FUNCTION_BLOCK Recipe_10054_FreePassion_special
VAR_INPUT
	execute: BOOL;
	Order: DUT_RECIPEORDER;
END_VAR
VAR_OUTPUT
	RecipeInfo: DUT_RECIPEOFFER;
	RecipeDone: BOOL;
	InitDone: BOOL;
END_VAR
VAR
	userparametersum: LREAL;
	StepDone: BOOL;
	i: INT;
END_VAR

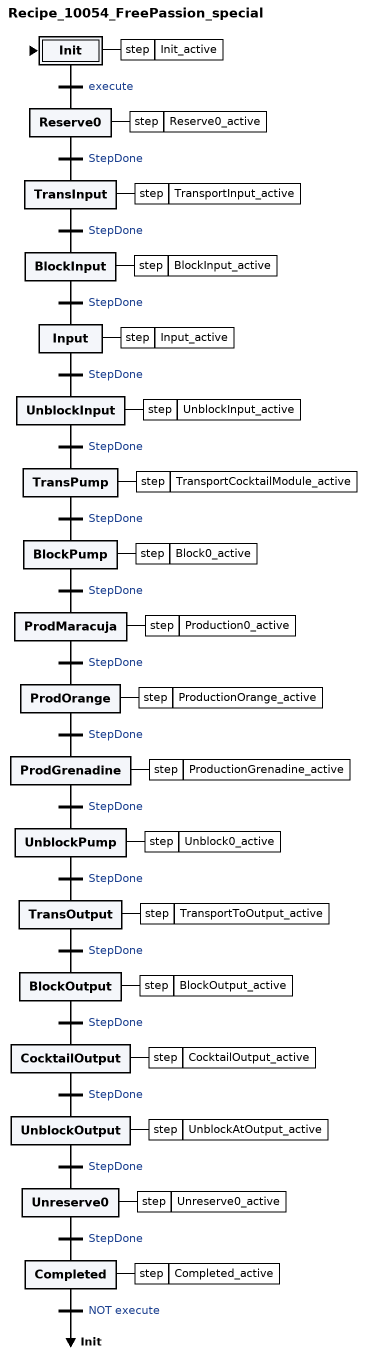
INITIAL_STEP Init:
    Init_active(N);  // step action
END_STEP
TRANSITION FROM Init TO Reserve0
    := execute;
END_TRANSITION
STEP Reserve0:
    Reserve0_active(N);  // step action
END_STEP
TRANSITION FROM Reserve0 TO TransInput
    := StepDone;
END_TRANSITION
STEP TransInput:
    TransportInput_active(N);  // step action
END_STEP
TRANSITION FROM TransInput TO BlockInput
    := StepDone;
END_TRANSITION
STEP BlockInput:
    BlockInput_active(N);  // step action
END_STEP
TRANSITION FROM BlockInput TO Input
    := StepDone;
END_TRANSITION
STEP Input:
    Input_active(N);  // step action
END_STEP
TRANSITION FROM Input TO UnblockInput
    := StepDone;
END_TRANSITION
STEP UnblockInput:
    UnblockInput_active(N);  // step action
END_STEP
TRANSITION FROM UnblockInput TO TransPump
    := StepDone;
END_TRANSITION
STEP TransPump:
    TransportCocktailModule_active(N);  // step action
END_STEP
TRANSITION FROM TransPump TO BlockPump
    := StepDone;
END_TRANSITION
STEP BlockPump:
    Block0_active(N);  // step action
END_STEP
TRANSITION FROM BlockPump TO ProdMaracuja
    := StepDone;
END_TRANSITION
STEP ProdMaracuja:
    Production0_active(N);  // step action
END_STEP
TRANSITION FROM ProdMaracuja TO ProdOrange
    := StepDone;
END_TRANSITION
STEP ProdOrange:
    ProductionOrange_active(N);  // step action
END_STEP
TRANSITION FROM ProdOrange TO ProdGrenadine
    := StepDone;
END_TRANSITION
STEP ProdGrenadine:
    ProductionGrenadine_active(N);  // step action
END_STEP
TRANSITION FROM ProdGrenadine TO UnblockPump
    := StepDone;
END_TRANSITION
STEP UnblockPump:
    Unblock0_active(N);  // step action
END_STEP
TRANSITION FROM UnblockPump TO TransOutput
    := StepDone;
END_TRANSITION
STEP TransOutput:
    TransportToOutput_active(N);  // step action
END_STEP
TRANSITION FROM TransOutput TO BlockOutput
    := StepDone;
END_TRANSITION
STEP BlockOutput:
    BlockOutput_active(N);  // step action
END_STEP
TRANSITION FROM BlockOutput TO CocktailOutput
    := StepDone;
END_TRANSITION
STEP CocktailOutput:
    CocktailOutput_active(N);  // step action
END_STEP
TRANSITION FROM CocktailOutput TO UnblockOutput
    := StepDone;
END_TRANSITION
STEP UnblockOutput:
    UnblockAtOutput_active(N);  // step action
END_STEP
TRANSITION FROM UnblockOutput TO Unreserve0
    := StepDone;
END_TRANSITION
STEP Unreserve0:
    Unreserve0_active(N);  // step action
END_STEP
TRANSITION FROM Unreserve0 TO Completed
    := StepDone;
END_TRANSITION
STEP Completed:
    Completed_active(N);  // step action
END_STEP
TRANSITION FROM Completed TO Init
    := NOT execute;
END_TRANSITION

ACTION Production0_active:
StepDone := FALSE;

userparametersum := 0;
FOR i := 1 TO UserParameterCnt DO
	IF NOT (order.UserParameter[i].Value = 0) THEN
		userparametersum := userparametersum + order.UserParameter[i].Value;
	
	END_IF
END_FOR
IF userparametersum = 0 THEN
userparametersum := -1;
END_IF
//Skill auswählen
ExecuteSkill.SkillID 		:= 1113;
ExecuteSkill.SkillName	 	:= 'Marajuca Juice';

//Parameter setzen

ExecuteSkill.Parameter[0].ID := 1;
ExecuteSkill.Parameter[0].Name := 'Quantity';
//order.userParameter[0] = amount
ExecuteSkill.Parameter[0].Value := order.UserParameter[0].Value * order.UserParameter[1].Value / userparametersum;//Summe aller Zutatenmengen;


(*
ExecuteSkill.Parameter[2].ID := ;
ExecuteSkill.Parameter[2].Name := '';
ExecuteSkill.Parameter[2].Value := ;
*)

(*
ExecuteSkill.Parameter[3].ID := ;
ExecuteSkill.Parameter[3].Name := '';
ExecuteSkill.Parameter[3].Value := ;
*)

(*
ExecuteSkill.Parameter[4].ID := ;
ExecuteSkill.Parameter[4].Name := '';
ExecuteSkill.Parameter[4].Value := ;
*)

(*
ExecuteSkill.Parameter[5].ID := ;
ExecuteSkill.Parameter[5].Name := '';
ExecuteSkill.Parameter[5].Value := ;
*)



ExecuteSkill();

StepDone := ExecuteSkill.Done;
END_ACTION

ACTION TransportInput_active:
StepDone := FALSE;

//Skill auswählen
ExecuteSkill.SkillID 		:= 1320;
ExecuteSkill.SkillName	 	:= 'Transport';

//Parameter setzen

ExecuteSkill.Parameter[3].ID := 3;
ExecuteSkill.Parameter[3].Name := 'Velocity';
ExecuteSkill.Parameter[3].Value := 1500;



ExecuteSkill.Parameter[1].ID :=  1;
ExecuteSkill.Parameter[1].Name := 'TargetPosition X';
ExecuteSkill.Parameter[1].Value := 30 ;
ExecuteSkill.Parameter[1].StringValue := '#DP#2#XPosition';



ExecuteSkill.Parameter[2].ID := 2;
ExecuteSkill.Parameter[2].Name := 'TargetPosition Z';
ExecuteSkill.Parameter[2].Value := 100;// ZCookieModule - ZCookieModuleCalibration - 2* Cookiethickness + toppingthickness+ Preasureheight  ;



(*
ExecuteSkill.Parameter[4].ID := 4;
ExecuteSkill.Parameter[4].Name := 'Acceleration';
ExecuteSkill.Parameter[4].Value := 0 ;
*)

(*
ExecuteSkill.Parameter[5].ID := ;
ExecuteSkill.Parameter[5].Name := '';
ExecuteSkill.Parameter[5].Value := ;
*)



ExecuteSkill();

StepDone := ExecuteSkill.Done;
END_ACTION

ACTION BlockOutput_active:
StepDone := FALSE;

//Skill auswählen
ExecuteSkill.SkillID 		:= 1315;
ExecuteSkill.SkillName	 	:= 'Block';

//Parameter setzen

ExecuteSkill.Parameter[1].ID := 1;
ExecuteSkill.Parameter[1].Name := 'TaskID';
ExecuteSkill.Parameter[1].Value := Order.TaskID;


(*
ExecuteSkill.Parameter[2].ID := ;
ExecuteSkill.Parameter[2].Name := '';
ExecuteSkill.Parameter[2].Value := ;
*)

(*
ExecuteSkill.Parameter[3].ID := ;
ExecuteSkill.Parameter[3].Name := '';
ExecuteSkill.Parameter[3].Value := ;
*)

(*
ExecuteSkill.Parameter[4].ID := ;
ExecuteSkill.Parameter[4].Name := '';
ExecuteSkill.Parameter[4].Value := ;
*)

(*
ExecuteSkill.Parameter[5].ID := ;
ExecuteSkill.Parameter[5].Name := '';
ExecuteSkill.Parameter[5].Value := ;
*)



ExecuteSkill();

StepDone := ExecuteSkill.Done;
END_ACTION

ACTION ProductionGrenadine_active:
StepDone := FALSE;

//Skill auswählen
ExecuteSkill.SkillID 		:= 1121;
ExecuteSkill.SkillName	 	:= 'Batida de Coco';

//Parameter setzen

ExecuteSkill.Parameter[0].ID := 1;
ExecuteSkill.Parameter[0].Name := 'Quantity';
//order.userParameter[0] = amount
ExecuteSkill.Parameter[0].Value := order.UserParameter[0].Value * order.UserParameter[3].Value / userparametersum; //Summe aller Zutatenmengen;



(*
ExecuteSkill.Parameter[2].ID := ;
ExecuteSkill.Parameter[2].Name := '';
ExecuteSkill.Parameter[2].Value := ;
*)

(*
ExecuteSkill.Parameter[3].ID := ;
ExecuteSkill.Parameter[3].Name := '';
ExecuteSkill.Parameter[3].Value := ;
*)

(*
ExecuteSkill.Parameter[4].ID := ;
ExecuteSkill.Parameter[4].Name := '';
ExecuteSkill.Parameter[4].Value := ;
*)

(*
ExecuteSkill.Parameter[5].ID := ;
ExecuteSkill.Parameter[5].Name := '';
ExecuteSkill.Parameter[5].Value := ;
*)



ExecuteSkill();

StepDone := ExecuteSkill.Done;
END_ACTION

ACTION Unreserve0_active:
StepDone := FALSE;

//Skill auswählen
ExecuteSkill.SkillID 		:= 1311;
ExecuteSkill.SkillName	 	:= 'Unreserve';

//Parameter setzen

ExecuteSkill.Parameter[1].ID := 1;
ExecuteSkill.Parameter[1].Name := 'TaskID';
ExecuteSkill.Parameter[1].Value := Order.TaskID;


(*
ExecuteSkill.Parameter[2].ID := ;
ExecuteSkill.Parameter[2].Name := '';
ExecuteSkill.Parameter[2].Val ue := ;
*)

(*
ExecuteSkill.Parameter[3].ID := ;
ExecuteSkill.Parameter[3].Name := '';
ExecuteSkill.Parameter[3].Value := ;
*)

(*
ExecuteSkill.Parameter[4].ID := ;
ExecuteSkill.Parameter[4].Name := '';
ExecuteSkill.Parameter[4].Value := ;
*)

(*
ExecuteSkill.Parameter[5].ID := ;
ExecuteSkill.Parameter[5].Name := '';
ExecuteSkill.Parameter[5].Value := ;
*)



ExecuteSkill();

StepDone := ExecuteSkill.Done;
END_ACTION

ACTION Input_active:
StepDone := FALSE;

//Skill auswählen
ExecuteSkill.SkillID 		:= 1402;
ExecuteSkill.SkillName	 	:= 'Input';

//Parameter setzen

ExecuteSkill.Parameter[1].ID := 1;
ExecuteSkill.Parameter[1].Name := 'TaskID';
ExecuteSkill.Parameter[1].Value := Order.TaskID;


(*
ExecuteSkill.Parameter[2].ID := ;
ExecuteSkill.Parameter[2].Name := '';
ExecuteSkill.Parameter[2].Value := ;
*)

(*
ExecuteSkill.Parameter[3].ID := ;
ExecuteSkill.Parameter[3].Name := '';
ExecuteSkill.Parameter[3].Value := ;
*)

(*
ExecuteSkill.Parameter[4].ID := ;
ExecuteSkill.Parameter[4].Name := '';
ExecuteSkill.Parameter[4].Value := ;
*)

(*
ExecuteSkill.Parameter[5].ID := ;
ExecuteSkill.Parameter[5].Name := '';
ExecuteSkill.Parameter[5].Value := ;
*)



ExecuteSkill();

StepDone := ExecuteSkill.Done;
END_ACTION

ACTION TransportToOutput_active:
StepDone := FALSE;

//Skill auswählen
ExecuteSkill.SkillID 		:= 1320;
ExecuteSkill.SkillName	 	:= 'Transport';

//Parameter setzen

ExecuteSkill.Parameter[3].ID := 3;
ExecuteSkill.Parameter[3].Name := 'Velocity';
ExecuteSkill.Parameter[3].Value := 280;



ExecuteSkill.Parameter[1].ID :=  1;
ExecuteSkill.Parameter[1].Name := 'TargetPosition X';
ExecuteSkill.Parameter[1].Value := 30 ;
ExecuteSkill.Parameter[1].StringValue := '#DP#2#XPosition';



ExecuteSkill.Parameter[2].ID := 2;
ExecuteSkill.Parameter[2].Name := 'TargetPosition Z';
ExecuteSkill.Parameter[2].Value := ZInputOutput;// ZCookieModule - ZCookieModuleCalibration - 2* Cookiethickness + toppingthickness+ Preasureheight  ;



(* ExecuteSkill.Parameter[4].ID := 4;
ExecuteSkill.Parameter[4].Name := 'Acceleration';
ExecuteSkill.Parameter[4].Value :=0 ;

*)
(*
ExecuteSkill.Parameter[5].ID := ;
ExecuteSkill.Parameter[5].Name := '';
ExecuteSkill.Parameter[5].Value := ;
*)



ExecuteSkill();

StepDone := ExecuteSkill.Done;
END_ACTION

ACTION ProductionOrange_active:
StepDone := FALSE;

//Skill auswählen
ExecuteSkill.SkillID 		:= 1117;
ExecuteSkill.SkillName	 	:= 'Orange';

//Parameter setzen

ExecuteSkill.Parameter[0].ID := 1;
ExecuteSkill.Parameter[0].Name := 'Quantity';
//order.userParameter[0] = amount
ExecuteSkill.Parameter[0].Value := order.UserParameter[0].Value * order.UserParameter[2].Value / userparametersum;//Summe aller Zutatenmengen;



(*
ExecuteSkill.Parameter[2].ID := ;
ExecuteSkill.Parameter[2].Name := '';
ExecuteSkill.Parameter[2].Value := ;
*)

(*
ExecuteSkill.Parameter[3].ID := ;
ExecuteSkill.Parameter[3].Name := '';
ExecuteSkill.Parameter[3].Value := ;
*)

(*
ExecuteSkill.Parameter[4].ID := ;
ExecuteSkill.Parameter[4].Name := '';
ExecuteSkill.Parameter[4].Value := ;
*)

(*
ExecuteSkill.Parameter[5].ID := ;
ExecuteSkill.Parameter[5].Name := '';
ExecuteSkill.Parameter[5].Value := ;
*)



ExecuteSkill();

StepDone := ExecuteSkill.Done;
END_ACTION

ACTION UnblockAtOutput_active:
StepDone := FALSE;

//Skill auswählen
ExecuteSkill.SkillID 		:= 1316;
ExecuteSkill.SkillName	 	:= 'Unblock';

//Parameter setzen

ExecuteSkill.Parameter[1].ID := 1;
ExecuteSkill.Parameter[1].Name := 'TaskID';
ExecuteSkill.Parameter[1].Value := Order.TaskID;


(*
ExecuteSkill.Parameter[2].ID := ;
ExecuteSkill.Parameter[2].Name := '';
ExecuteSkill.Parameter[2].Value := ;
*)

(*
ExecuteSkill.Parameter[3].ID := ;
ExecuteSkill.Parameter[3].Name := '';
ExecuteSkill.Parameter[3].Value := ;
*)

(*
ExecuteSkill.Parameter[4].ID := ;
ExecuteSkill.Parameter[4].Name := '';
ExecuteSkill.Parameter[4].Value := ;
*)

(*
ExecuteSkill.Parameter[5].ID := ;
ExecuteSkill.Parameter[5].Name := '';
ExecuteSkill.Parameter[5].Value := ;
*)



ExecuteSkill();

StepDone := ExecuteSkill.Done;
END_ACTION

ACTION CocktailOutput_active:
StepDone := FALSE;

//Skill auswählen
ExecuteSkill.SkillID 		:= 1403;
ExecuteSkill.SkillName	 	:= 'Output';

//Parameter setzen

ExecuteSkill.Parameter[1].ID := 1;
ExecuteSkill.Parameter[1].Name := 'TaskID';
ExecuteSkill.Parameter[1].Value := Order.TaskID;


(*
ExecuteSkill.Parameter[2].ID := ;
ExecuteSkill.Parameter[2].Name := '';
ExecuteSkill.Parameter[2].Value := ;
*)

(*
ExecuteSkill.Parameter[3].ID := ;
ExecuteSkill.Parameter[3].Name := '';
ExecuteSkill.Parameter[3].Value := ;
*)

(*
ExecuteSkill.Parameter[4].ID := ;
ExecuteSkill.Parameter[4].Name := '';
ExecuteSkill.Parameter[4].Value := ;
*)

(*
ExecuteSkill.Parameter[5].ID := ;
ExecuteSkill.Parameter[5].Name := '';
ExecuteSkill.Parameter[5].Value := ;
*)

ExecuteSkill();

StepDone := ExecuteSkill.Done;
END_ACTION

ACTION Completed_active:
RecipeDone := TRUE;
StepDone := FALSE;
END_ACTION

ACTION UnblockInput_active:
StepDone := FALSE;

//Skill auswählen
ExecuteSkill.SkillID 		:= 1316;
ExecuteSkill.SkillName	 	:= 'Unblock';

//Parameter setzen

ExecuteSkill.Parameter[1].ID := 1;
ExecuteSkill.Parameter[1].Name := 'TaskID';
ExecuteSkill.Parameter[1].Value := Order.TaskID;


(*
ExecuteSkill.Parameter[2].ID := ;
ExecuteSkill.Parameter[2].Name := '';
ExecuteSkill.Parameter[2].Value := ;
*)

(*
ExecuteSkill.Parameter[3].ID := ;
ExecuteSkill.Parameter[3].Name := '';
ExecuteSkill.Parameter[3].Value := ;
*)

(*
ExecuteSkill.Parameter[4].ID := ;
ExecuteSkill.Parameter[4].Name := '';
ExecuteSkill.Parameter[4].Value := ;
*)

(*
ExecuteSkill.Parameter[5].ID := ;
ExecuteSkill.Parameter[5].Name := '';
ExecuteSkill.Parameter[5].Value := ;
*)



ExecuteSkill();

StepDone := ExecuteSkill.Done;
END_ACTION

ACTION Unblock0_active:
StepDone := FALSE;

//Skill auswählen
ExecuteSkill.SkillID 		:= 1316;
ExecuteSkill.SkillName	 	:= 'Unblock';

//Parameter setzen

ExecuteSkill.Parameter[1].ID := 1;
ExecuteSkill.Parameter[1].Name := 'TaskID';
ExecuteSkill.Parameter[1].Value := Order.TaskID;


(*
ExecuteSkill.Parameter[2].ID := ;
ExecuteSkill.Parameter[2].Name := '';
ExecuteSkill.Parameter[2].Value := ;
*)

(*
ExecuteSkill.Parameter[3].ID := ;
ExecuteSkill.Parameter[3].Name := '';
ExecuteSkill.Parameter[3].Value := ;
*)

(*
ExecuteSkill.Parameter[4].ID := ;
ExecuteSkill.Parameter[4].Name := '';
ExecuteSkill.Parameter[4].Value := ;
*)

(*
ExecuteSkill.Parameter[5].ID := ;
ExecuteSkill.Parameter[5].Name := '';
ExecuteSkill.Parameter[5].Value := ;
*)



ExecuteSkill();

StepDone := ExecuteSkill.Done;
END_ACTION

ACTION TransportCocktailModule_active:
StepDone := FALSE;

//Skill auswählen
ExecuteSkill.SkillID 		:= 1320;
ExecuteSkill.SkillName	 	:= 'Transport';

//Parameter setzen

ExecuteSkill.Parameter[3].ID := 3;
ExecuteSkill.Parameter[3].Name := 'Velocity';
ExecuteSkill.Parameter[3].Value := 1000;



ExecuteSkill.Parameter[1].ID :=  1;
ExecuteSkill.Parameter[1].Name := 'TargetPosition X';
ExecuteSkill.Parameter[1].Value := 30 ;
ExecuteSkill.Parameter[1].StringValue := '#DP#2#XPosition';



ExecuteSkill.Parameter[2].ID := 2;
ExecuteSkill.Parameter[2].Name := 'TargetPosition Z';
ExecuteSkill.Parameter[2].Value := 40;// ZCookieModule - ZCookieModuleCalibration - 2* Cookiethickness + toppingthickness+ Preasureheight  ;



(*
ExecuteSkill.Parameter[4].ID := 4;
ExecuteSkill.Parameter[4].Name := 'Acceleration';
ExecuteSkill.Parameter[4].Value := 0 ;
*)

(*
ExecuteSkill.Parameter[5].ID := ;
ExecuteSkill.Parameter[5].Name := '';
ExecuteSkill.Parameter[5].Value := ;
*)



ExecuteSkill();

StepDone := ExecuteSkill.Done;
END_ACTION

ACTION Init_active:
RecipeDone := FALSE;

// Initialisation of Recipe Parameters an name etc
RecipeInfo.Name := 'Free Passion special';
RecipeInfo.Description := 'Sweet cocktail combining the sourness of maracuja and orange juice with the taste of Coco';
RecipeInfo.Dummy := FALSE;
RecipeInfo.RecipeID := 10054; 	// 
Initdone := TRUE;

FOR i := 0 TO UserParameterCnt DO
	IF Order.UserParameter[i].Value = 0 THEN
		order.UserParameter[i].Value := RecipeInfo.UserParameter[i].Default;
	END_IF
END_FOR
//Parameter 0:

	RecipeInfo.UserParameter[0].Dummy 		:= FALSE;
	RecipeInfo.UserParameter[0].Default		:= 200;
	RecipeInfo.UserParameter[0].Description	:= 'Gives the total fluid amount in the glass';
	RecipeInfo.UserParameter[0].MaxValue	:= 200;
	RecipeInfo.UserParameter[0].MinValue	:= 10;
	RecipeInfo.UserParameter[0].Name		:= 'Total Liquid Amount';
	RecipeInfo.UserParameter[0].Unit		:= 'ml';
	
//Parameter 1:

	RecipeInfo.UserParameter[1].Dummy 		:= FALSE;
	RecipeInfo.UserParameter[1].Default		:= 50;
	RecipeInfo.UserParameter[1].Description	:= 'Maracuja Juice';
	RecipeInfo.UserParameter[1].MaxValue	:= 100;
	RecipeInfo.UserParameter[1].MinValue	:= 1;
	RecipeInfo.UserParameter[1].Name		:= 'Maracuja Juice';
	RecipeInfo.UserParameter[1].Unit		:= 'ml';
	
//Parameter 2:

	RecipeInfo.UserParameter[2].Dummy 		:= FALSE;
	RecipeInfo.UserParameter[2].Default		:= 35;
	RecipeInfo.UserParameter[2].Description	:= 'Orange Juice';
	RecipeInfo.UserParameter[2].MaxValue	:= 100;
	RecipeInfo.UserParameter[2].MinValue	:= 1;
	RecipeInfo.UserParameter[2].Name		:= 'Orange Juice';
	RecipeInfo.UserParameter[2].Unit		:= 'ml';

//Parameter 3:

	RecipeInfo.UserParameter[3].Dummy 		:= FALSE;
	RecipeInfo.UserParameter[3].Default		:= 15;
	RecipeInfo.UserParameter[3].Description	:= 'Batida de Coco';
	RecipeInfo.UserParameter[3].MaxValue	:= 50;
	RecipeInfo.UserParameter[3].MinValue	:= 1;
	RecipeInfo.UserParameter[3].Name		:= 'Batida de Coco';
	RecipeInfo.UserParameter[3].Unit		:= 'ml';
	
	
	
//Parameter 1:
(*
	RecipeInfo.UserParameter[1].Dummy 		:= 
	RecipeInfo.UserParameter[1].Default		:=
	RecipeInfo.UserParameter[1].Description	:=
	RecipeInfo.UserParameter[1].MaxValue	:=
	RecipeInfo.UserParameter[1].MinValue	:=
	RecipeInfo.UserParameter[1].Name		:=
	RecipeInfo.UserParameter[1].Unit		:=
*)
//Parameter 2:

(*
	RecipeInfo.UserParameter[2].Dummy 		:= 
	RecipeInfo.UserParameter[2].Default		:=
	RecipeInfo.UserParameter[2].Description	:=
	RecipeInfo.UserParameter[2].MaxValue	:=
	RecipeInfo.UserParameter[2].MinValue	:=
	RecipeInfo.UserParameter[2].Name		:=
	RecipeInfo.UserParameter[2].Unit		:=
*)

//Parameter 3:

(*
	RecipeInfo.UserParameter[3].Dummy 		:= 
	RecipeInfo.UserParameter[3].Default		:=
	RecipeInfo.UserParameter[3].Description	:=
	RecipeInfo.UserParameter[3].MaxValue	:=
	RecipeInfo.UserParameter[3].MinValue	:=
	RecipeInfo.UserParameter[3].Name		:=
	RecipeInfo.UserParameter[3].Unit		:=
*)

//Parameter 4:

(*
	RecipeInfo.UserParameter[4].Dummy 		:= 
	RecipeInfo.UserParameter[4].Default		:=
	RecipeInfo.UserParameter[4].Description	:=
	RecipeInfo.UserParameter[4].MaxValue	:=
	RecipeInfo.UserParameter[4].MinValue	:=
	RecipeInfo.UserParameter[4].Name		:=
	RecipeInfo.UserParameter[4].Unit		:=
*)


//Parameter 5:

(*
	RecipeInfo.UserParameter[5].Dummy 		:= 
	RecipeInfo.UserParameter[5].Default		:=
	RecipeInfo.UserParameter[5].Description	:=
	RecipeInfo.UserParameter[5].MaxValue	:=
	RecipeInfo.UserParameter[5].MinValue	:=
	RecipeInfo.UserParameter[5].Name		:=
	RecipeInfo.UserParameter[5].Unit		:=
*)
END_ACTION

ACTION Block0_active:
StepDone := FALSE;

//Skill auswählen
ExecuteSkill.SkillID 		:= 1315;
ExecuteSkill.SkillName	 	:= 'Block';

//Parameter setzen

ExecuteSkill.Parameter[1].ID := 1;
ExecuteSkill.Parameter[1].Name := 'TaskID';
ExecuteSkill.Parameter[1].Value := Order.TaskID;


(*
ExecuteSkill.Parameter[2].ID := ;
ExecuteSkill.Parameter[2].Name := '';
ExecuteSkill.Parameter[2].Value := ;
*)

(*
ExecuteSkill.Parameter[3].ID := ;
ExecuteSkill.Parameter[3].Name := '';
ExecuteSkill.Parameter[3].Value := ;
*)

(*
ExecuteSkill.Parameter[4].ID := ;
ExecuteSkill.Parameter[4].Name := '';
ExecuteSkill.Parameter[4].Value := ;
*)

(*
ExecuteSkill.Parameter[5].ID := ;
ExecuteSkill.Parameter[5].Name := '';
ExecuteSkill.Parameter[5].Value := ;
*)



ExecuteSkill();

StepDone := ExecuteSkill.Done;
END_ACTION

ACTION Reserve0_active:
StepDone := FALSE;
RecipeDone := FALSE;
//Skill auswählen
ExecuteSkill.SkillID 		:= 1310;
ExecuteSkill.SkillName	 	:= 'Reserve';

//Parameter setzen

ExecuteSkill.Parameter[1].ID := 1;
ExecuteSkill.Parameter[1].Name := 'TaskID';
ExecuteSkill.Parameter[1].Value := Order.TaskID;


(*
ExecuteSkill.Parameter[2].ID := ;
ExecuteSkill.Parameter[2].Name := '';
ExecuteSkill.Parameter[2].Value := ;
*)

(*
ExecuteSkill.Parameter[3].ID := ;
ExecuteSkill.Parameter[3].Name := '';
ExecuteSkill.Parameter[3].Value := ;
*)

(*
ExecuteSkill.Parameter[4].ID := ;
ExecuteSkill.Parameter[4].Name := '';
ExecuteSkill.Parameter[4].Value := ;
*)

(*
ExecuteSkill.Parameter[5].ID := ;
ExecuteSkill.Parameter[5].Name := '';
ExecuteSkill.Parameter[5].Value := ;
*)



ExecuteSkill();

StepDone := ExecuteSkill.Done;
END_ACTION

ACTION BlockInput_active:
StepDone := FALSE;

//Skill auswählen
ExecuteSkill.SkillID 		:= 1315;
ExecuteSkill.SkillName	 	:= 'Block';

//Parameter setzen

ExecuteSkill.Parameter[1].ID := 1;
ExecuteSkill.Parameter[1].Name := 'TaskID';
ExecuteSkill.Parameter[1].Value := Order.TaskID;


(*
ExecuteSkill.Parameter[2].ID := ;
ExecuteSkill.Parameter[2].Name := '';
ExecuteSkill.Parameter[2].Value := ;
*)

(*
ExecuteSkill.Parameter[3].ID := ;
ExecuteSkill.Parameter[3].Name := '';
ExecuteSkill.Parameter[3].Value := ;
*)

(*
ExecuteSkill.Parameter[4].ID := ;
ExecuteSkill.Parameter[4].Name := '';
ExecuteSkill.Parameter[4].Value := ;
*)

(*
ExecuteSkill.Parameter[5].ID := ;
ExecuteSkill.Parameter[5].Name := '';
ExecuteSkill.Parameter[5].Value := ;
*)



ExecuteSkill();

StepDone := ExecuteSkill.Done;
END_ACTION

END_FUNCTION_BLOCK

(* stored: Version 1.1.0.1, ProductVersion 3.1.0.25
   POU Recipe_10054_FreePassion_special: Id {a4817f5a-9739-4444-b53b-f9e469c50c3a}
   Action Production0_active: Id {00f65884-65f7-4ac0-9903-73cbb35c8302}
   Action TransportInput_active: Id {075bc388-bf80-4e1c-b9b6-9227c2a19d9c}
   Action BlockOutput_active: Id {084309fc-f299-4671-87cd-b855609607fb}
   Action ProductionGrenadine_active: Id {1007c1c0-d427-4d3e-80d8-1052fef8cd39}
   Action Unreserve0_active: Id {1698fc29-a372-4fde-adf1-ab718e1278f2}
   Action Input_active: Id {6ebc2a18-723c-45ea-bedf-cc7342ebe416}
   Action TransportToOutput_active: Id {6f9ae2fa-52ee-4dce-a3e1-afa17f1b3283}
   Action ProductionOrange_active: Id {754652cf-b042-4beb-819e-95b98bbb9c70}
   Action UnblockAtOutput_active: Id {99f7c574-8815-472f-be9c-9749d9548ee8}
   Action CocktailOutput_active: Id {9aabe13d-48a9-4515-8734-a1ce9c97a838}
   Action Completed_active: Id {b3b2285f-77fa-4913-80cd-3472d49b1e16}
   Action UnblockInput_active: Id {bae56393-0d06-46ed-9ed9-ffc99813ef55}
   Action Unblock0_active: Id {c4ee4e0f-d582-41c1-98d8-7e54118d0306}
   Action TransportCocktailModule_active: Id {eeb02142-7f29-437d-9b77-7b32b44b409e}
   Action Init_active: Id {f2501569-911a-4108-8a97-3838bda174e6}
   Action Block0_active: Id {f6acfd2a-131f-4a34-b685-bb17b9dd9be3}
   Action Reserve0_active: Id {f854676d-c9a2-48e6-88fa-acff07d071c5}
   Action BlockInput_active: Id {fe999b71-ed6f-4d89-8ecd-f46b4b284f84} *)
